{attribute 'linkalways'} 
{attribute 'no_explicit_call' := 'This FB is a CLASS and must be accessed using methods or properties'}
{attribute 'enable_dynamic_creation'}
FUNCTION_BLOCK ABSTRACT NciCommand EXTENDS Command IMPLEMENTS I_NciCommand

END_FUNCTION_BLOCK

(* stored: Version 1.1.0.1, ProductVersion 3.1.4024.12
   POU NciCommand: Id {4a3ff4ae-a914-42b7-9d67-a7b8c3276d0a}, SpecialFunc None *)
